ABB RobotStudio station: Práctica5_inicio.rspag

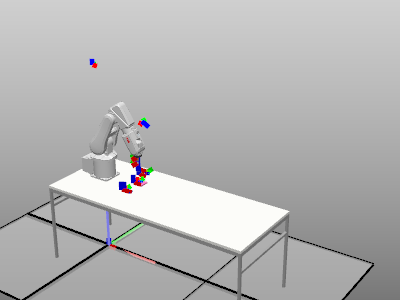
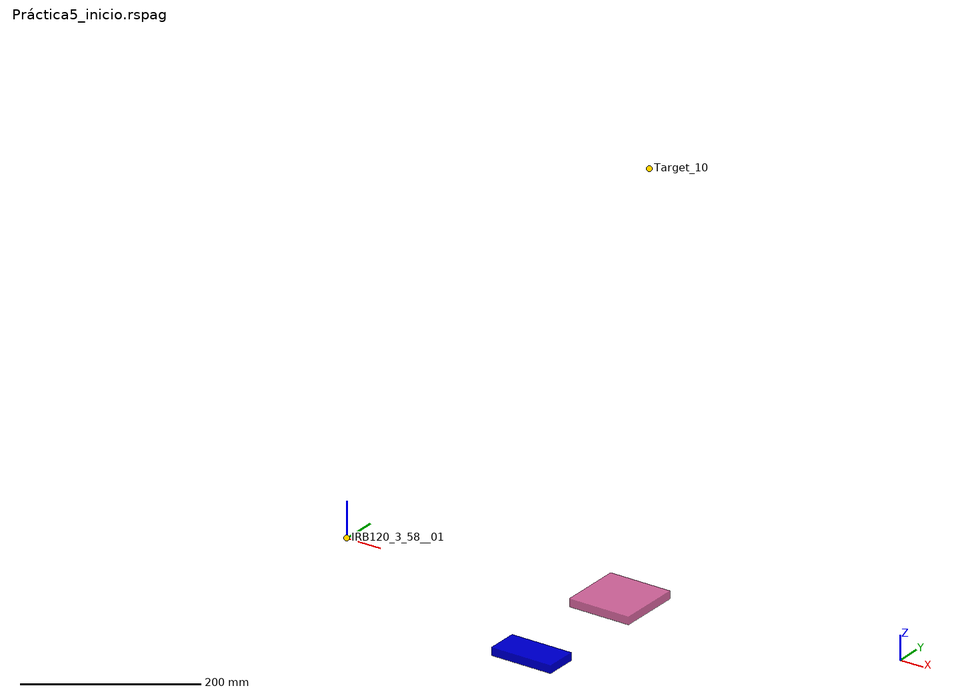
[picture v1: parts stored in the station drawn from their meshes, with robot base, taught points and paths (robot models come from the ABB library and are not in the file)]
--- station ---
Station Práctica3_inicio (saved by RobotStudio 25.1.11133.0)
Controller Controlador2, task T_ROB1: task frame (RAPID world) sits at (0, 0, 670) mm in the station
Controller Controlador2
  mechanical unit ROB_1: IRB120_3_58__01, 6 joints, base frame (0, 0, 0) mm
Layout (positions relative to the parent item):
  - TVentosa [mechanism] at (320, 40, 901.19) mm, rotated rx -180 ry 0 rz -90 deg
      TCP TVentosa at (0, 0, 51.19) mm
      links: Mi_herramienta
  - LogicGate [smart component, from Components\LogicGate.rslib]
      properties: Operator=NOT; Delay=0
  - LogicGate_2 [smart component, from Components\LogicGate.rslib]
      properties: Operator=AND; Delay=0
  - IRB120_3_58__01 [mechanism, from %ABB.RobotStudio.Models.IRB120%\IRB120_3_58_G_01.rslib] at (0, 0, 670) mm; joint values [0.1244, 0.4423, 0.6254, 0, 0.5031, -1.4464] (rad or m)
  - table [part, from Libraries\e293a11e-ed86-4237-866f-a9bf8f4bd145table.rslib] at (-246.62, 300, 670) mm, rotated rx 0 ry 0 rz -90 deg
  - Base2 [part], size 80 x 80 x 10 mm
  - Base1 [part], size 80 x 40 x 10 mm
  - Detacher [smart component, from Components\Detacher.rslib]
      properties: Child=Link6; KeepPosition=true
  - CollisionSensor [smart component, from Components\CollisionSensor.rslib]
      properties: Object1=TVentosa; Object2=(none); NearMiss=0.007; Part1=Mi_herramienta; Part2=Link6; CollisionType=1
    - _sensorPart_ [part]
  - Attacher_2 [smart component, from Components\Attacher.rslib]
      properties: Parent=TVentosa; Flange=0; Child=Link6; Mount=false; Offset=[0 0 0]; Orientation=[0 0 0]
  - Source_2 [smart component, from Components\Source.rslib]
      properties: Source=Pieza; Copy=(none); Parent=(none); Position=[0.34 -0.13 0.68]; Orientation=[0 0 0]; Transient=true; PhysicsBehavior=0
  - SimulationEvents_2 [smart component, from Components\SimulationEvents.rslib]
  - Pieza [part] at (340, -130, 700) mm, rotated rx 180 ry 0 rz 180 deg, size 60 x 20 x 20 mm
Attachment: TVentosa is attached to IRB120_3_58__01 / Link6
Attachment: Base2 is attached to Base1
Attachment: Base1 is attached to table
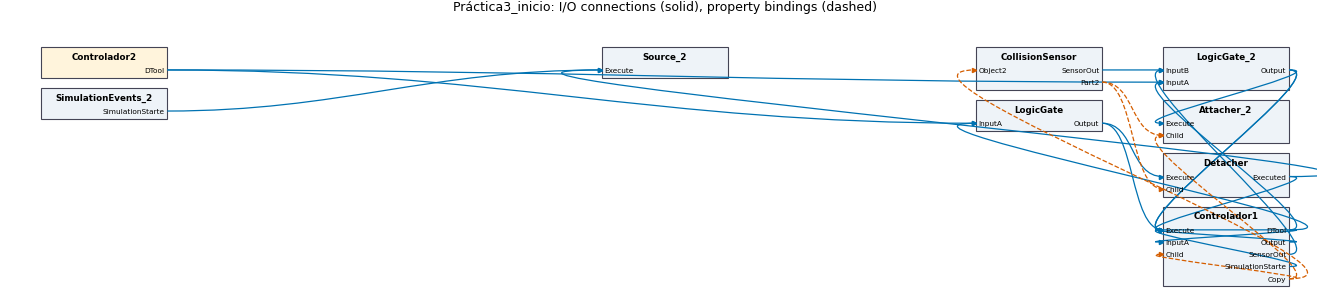
Station logic (signal -> signal, property => property):
  Controlador1.DTool -> Attacher.Execute
  Controlador1.DTool -> LogicGate_2.InputA
  LogicGate_2.Output -> Detacher.Execute
  Controlador1.DTool -> LogicGate.InputA
  LogicGate.Output -> Detacher.Execute
  CollisionSensor.SensorOut -> LogicGate_2.InputB
  Controlador1.DTool -> LogicGate_2.InputA
  LogicGate_2.Output -> Attacher.Execute
  Controlador2.DTool -> LogicGate.InputA
  LogicGate.Output -> Detacher.Execute
  Controlador2.DTool -> LogicGate_2.InputA
  LogicGate_2.Output -> Attacher.Execute
  Detacher.Executed -> Source.Execute
  SimulationEvents.SimulationStarted -> Source.Execute
  CollisionSensor.SensorOut -> LogicGate_2.InputB
  SimulationEvents_2.SimulationStarted -> Source_2.Execute
  Detacher.Executed -> Source_2.Execute
  LogicGate_2.Output -> Attacher_2.Execute
  Source.Copy => Attacher.Child
  Source.Copy => CollisionSensor.Object2
  Source.Copy => Attacher_2.Child
  CollisionSensor.Part2 => Detacher.Child
  CollisionSensor.Part2 => Attacher_2.Child
Targets, tools, work objects and paths stored in the station and not in the controller backup, written as RAPID:
! task T_ROB1
MODULE CalibData
  PROC Path_10()
    MoveJ Target_10,v200,z100,TVentosa\WObj:=wobj0;
    MoveL Target_20,v200,fine,TVentosa\WObj:=WO_Pieza;
    MoveL Target_30,v200,z100,TVentosa\WObj:=WO_Base2;
    MoveAbsJ JHome,v1000,z100,TVentosa\WObj:=WO_Pieza;
  ENDPROC
ENDMODULE

! task T_ROB1
MODULE Module1
  PROC Path_20()
    MoveJ Target_40,v1000,z100,TVentosa\WObj:=CajonDesastre;
  ENDPROC
ENDMODULE


--- Backups/Controlador2/RAPID/TASK1/PROGMOD/CalibData.mod ---
MODULE CalibData
    TASK PERS wobjdata Workobject_1:=[FALSE,TRUE,"",[[237.224,146.16,10],[1,0,0,0]],[[50,50,20],[0,0,1,0]]];
    TASK PERS wobjdata CajonDesastre:=[FALSE,TRUE,"",[[237.224,146.16,10],[1,0,0,0]],[[50,50,20],[0,0,1,0]]];
    PERS tooldata TVentosa:=[TRUE,[[0,0,51.19],[1,0,0,0]],[0.1,[0,0,1],[1,0,0,0],0,0,0]];
    TASK PERS wobjdata WO_Pieza:=[FALSE,TRUE,"",[[300,-150,10],[1,0,0,0]],[[20,10,0],[1,0,0,0]]];
    TASK PERS wobjdata WO_Base2:=[FALSE,TRUE,"",[[300,-150,10],[1,0,0,0]],[[0,150,0],[1,0,0,0]]];




ENDMODULE

--- Backups/Controlador2/RAPID/TASK1/PROGMOD/Module1.mod ---
MODULE Module1
    CONST robtarget Target_10:=[[408.685,0,568.405],[0.5,0,0.866025404,0],[0,0,0,0],[9E+09,9E+09,9E+09,9E+09,9E+09,9E+09]];
    CONST robtarget Target_20:=[[19.999989664,10.000006428,19.999948885],[-0.000000013,0,1,0.000000005],[-1,0,-1,0],[9E+09,9E+09,9E+09,9E+09,9E+09,9E+09]];
    CONST robtarget Target_30:=[[40,40,20],[0,0,1,0],[0,0,0,0],[9E+09,9E+09,9E+09,9E+09,9E+09,9E+09]];
    VAR num h;
    VAR num h_pieza:=20;
    CONST jointtarget JHome:=[[0,0,-90,0,0,0],[9E+09,9E+09,9E+09,9E+09,9E+09,9E+09]];
    VAR num pos_torre;
    VAR num Px;
    VAR num Py;
    VAR num Pz;
    VAR num Rz;
    VAR num pos;
    VAR robtarget punto_orig;
    VAR robtarget punto_dest;
    VAR num num_pieza;
    VAR num a;
    VAR num b;
    VAR num c;
    VAR num contador4;
    VAR num contador5;
    VAR num plantas_puestas;
    VAR num plantas_totales;
    VAR num planta;
    VAR num apartado;
    CONST robtarget Target_40:=[[0,0,0],[1,0,0,0],[0,0,0,0],[9E+09,9E+09,9E+09,9E+09,9E+09,9E+09]];
    !***********************************************************
    !
    ! Módulo:  Module1
    !
    ! Descripción:
    !   <Introduzca la descripción aquí>
    !
    ! Autor: Juan
    !
    ! Versión: 1.0
    !
    !***********************************************************

    PROC main()
        !Añada aquí su código
        Initialize;
        MoveJ Target_10,v1000,z100,TVentosa\WObj:=wobj0;
        WHILE DFin=0 DO
            IF DPieza=1 THEN
                !TPReadNum apartado,"¿Apartado en el que trabajamos? ()";
                apartado:=1;
                IF apartado=0 THEN
                    TPReadNum planta,"¿Número de plantas hasta el que quieres llegar? ()";
                    num_pieza:=planta*4;
                    a:=0;
                    b:=0;
                    a:=num_pieza DIV 4;
                    b:=num_pieza MOD 4;
                    IF a>0 THEN
                        FOR contador2 FROM 1 TO a DO
                            FOR contador FROM 0 TO 3 DO
                                Pick Target_20,WO_pieza;
                                Place Offs(calcula_posicion(contador),0,0,0),WO_Base2;
                                IF (contador=3) THEN
                                    h:=h+2*h_pieza;
                                ENDIF
                            ENDFOR
                        ENDFOR
                    ENDIF
                    IF b>0 THEN
                        FOR contador3 FROM 1 TO b DO
                            Pick Target_20,WO_pieza;
                            Place Offs(calcula_posicion(contador3-1),0,0,0),WO_Base2;
                            IF (contador3=3) THEN
                                h:=h+2*h_pieza;
                            ENDIF
                        ENDFOR
                    ENDIF
                ENDIF
                !APARTADO A
                !FOR contador4 FROM 1 TO num_pieza DO
                !   FOR contador5 FROM 1 TO 4 DO
                !        Pick Target_20, WO_pieza;
                !         Place(Offs(calcula_posicion(contador5 - 1),0,0,0));
                !       IF (contador5 =4) THEN
                !            h := h + 2*h_pieza;
                !        ENDIF
                !   ENDFOR
                !ENDFOR
                !preguntar como terminar el programa
                !******************************************
                !FOR contador5 FROM 1 TO 4 DO
                !               Pick Target_20,WO_pieza;
                !                Place(Offs(calcula_posicion(contador5-1),0,0,0));
                !               pos := contador5-1;
                !               IF (contador5=4) THEN
                !                   h:=h+2*h_pieza;
                !                   plantas_puestas:=plantas_puestas+1;
                !               ENDIF
                !           ENDFOR

                !*************************************************
                !APARTADO B
                IF apartado=1 THEN
                    TPReadNum planta,"¿Número de plantas hasta el que quieres llegar? ()";
                    plantas_totales:=planta-plantas_puestas;
                    IF plantas_totales>0 THEN
                        FOR contador4 FROM 4*plantas_puestas TO (4*planta)-1 DO
                            Pick Target_20,WO_pieza;
                            MoveL Offs(Target_20,0,0,50+5*contador4),v1000,z100,TVentosa\WObj:=WO_Pieza;
                            Place Offs(calcula_posicion(contador4),0,0,0),WO_Base2;
                            IF ((contador4+1) MOD 4)=0 THEN
                                plantas_puestas:=(contador4+1) DIV 4;
                            ENDIF
                        ENDFOR
                    ENDIF
                    IF plantas_totales<0 THEN
                        FOR contador6 FROM (4*plantas_puestas)-1 TO (-(4*plantas_totales)) DO

                            Pick calcula_posicion(contador6),WO_Base2;
                            Place Offs(Target_30,150,-200,100),WO_Base2;
                            IF ((contador6+1) MOD 4)=0 THEN
                                plantas_puestas:=(contador6) DIV 4;
                            ENDIF

                        ENDFOR

                        !h:=h-2*h_pieza;

                    ENDIF

                ENDIF

            ENDIF

        ENDWHILE
        MoveAbsJ JHome,v150,z200,TVentosa\WObj:=WO_Pieza;

    ENDPROC

    PROC Initialize()
        h:=0;
        pos_torre:=0;
        plantas_puestas:=0;
        plantas_totales:=0;
        a:=0;
        b:=0;
        c:=0;
        num_pieza:=0;
        planta:=0;
        apartado:=0;
    ENDPROC

    FUNC robtarget calcula_posicion(num planta)

        a:=planta DIV 4;
        b:=planta MOD 4;

        TEST b
        CASE 0:
            Px:=0;
            Py:=20;
            Pz:=-2*h_pieza*a;

            Rz:=0;
        CASE 1:
            Px:=0;
            Py:=-20;
            Pz:=-2*h_pieza*a;

            Rz:=0;

        CASE 2:
            Px:=-20;
            Py:=0;
            Pz:=-(2*h_pieza*a+h_pieza);

            Rz:=90;
        CASE 3:
            Px:=20;
            Py:=0;
            Pz:=-(2*h_pieza*a+h_pieza);

            Rz:=-90;
        DEFAULT:
        ENDTEST

        punto_orig:=Target_30;
        punto_dest:=RelTool(punto_orig,Px,Py,Pz\Rx:=0,\Ry:=0,\Rz:=Rz);
        RETURN punto_dest;

        !RelTool(Target_30,Px,Py,Pz \Rx := 0 \Ry := 0 \Rz := Rz);

    ENDFUNC

    PROC Pick(robtarget posicion,PERS wobjdata WO)
        MoveL Offs(posicion,0,0,50),v1000,z100,TVentosa\WObj:=WO;
        MoveL posicion,v1000,fine,TVentosa\WObj:=WO;
        SetDO DTool,1;
        MoveL Offs(posicion,0,0,50),v1000,z100,TVentosa\WObj:=WO;
    ENDPROC

    PROC Place(robtarget posicion,PERS wobjdata WO)
        MoveL Offs(posicion,0,0,50),v1000,fine,TVentosa\WObj:=WO;
        MoveL posicion,v1000,fine,TVentosa\WObj:=WO;
        SetDO DTool,0;
        MoveL Offs(posicion,0,0,50),v1000,fine,TVentosa\WObj:=WO;
    ENDPROC


ENDMODULE

--- Backups/Controlador2/SYSPAR/EIO.cfg ---
EIO:CFG_1.0:6:1::
#
EIO_SIGNAL:

      -Name "DFin" -SignalType "DI"

      -Name "DTool" -SignalType "DO"

      -Name "DPieza" -SignalType "DI"
